(* CoDeSys 2.3.9.31 project: 3floor7(20131104).prx *)
(* Libraries: TcEIB.lbx 31.10.12 09:33:08, TcBaseBX.lbx 10.5.06 08:50:20, TcSystemBX.lbx 11.6.12 13:56:16, standard.lbx 5.12.03 08:02:30 *)

(* Task configuration *)
TASK Standard (PRIORITY := 0, INTERVAL := T#20ms);
	MAIN
END_TASK

(* Global variable list: main *)
VAR_GLOBAL


	bDarkOutside: BOOL;
	fb_KL6301_0: KL6301; (* EIB functonblock *)


	VITALNYA_HVAC: ROOM_HVAC;
	SPALNYA_HVAC: ROOM_HVAC;
	DYTJACHA_HVAC: ROOM_HVAC;
	KINO_HVAC:ROOM_HVAC;
	STUDIO_HVAC: ROOM_HVAC;
	KABINET_HVAC:ROOM_HVAC;

(*adresses for Temperatures from HDL panels *)
	vitalnya_T_EIB_addr: EIB_GROUP_ADDR:= (MAIN:=1, SUB_MAIN:=1, NUMBER:=0);
	kino_T_EIB_addr: EIB_GROUP_ADDR:= (MAIN:=1, SUB_MAIN:=2, NUMBER:=0);
	studio_T_EIB_addr: EIB_GROUP_ADDR:= (MAIN:=1, SUB_MAIN:=3, NUMBER:=0);
	kabinet_T_EIB_addr: EIB_GROUP_ADDR:= (MAIN:=1, SUB_MAIN:=4, NUMBER:=0);
	dytjacha_T_EIB_addr: EIB_GROUP_ADDR:= (MAIN:=1, SUB_MAIN:=5, NUMBER:=0);
	spalnya_T_EIB_addr: EIB_GROUP_ADDR:= (MAIN:=1, SUB_MAIN:=6, NUMBER:=0);
(*adresses for current speed and setpoint of cooling mode from HDL panels *)
	dytjacha_cooling_EIB_addr: EIB_GROUP_ADDR:= (MAIN:=1, SUB_MAIN:=1, NUMBER:=1);
	spalnya_cooling_EIB_addr: EIB_GROUP_ADDR:= (MAIN:=1, SUB_MAIN:=2, NUMBER:=1);
	vitalnya_cooling_EIB_addr: EIB_GROUP_ADDR:= (MAIN:=1, SUB_MAIN:=3, NUMBER:=1);
	kino_cooling_EIB_addr: EIB_GROUP_ADDR:= (MAIN:=1, SUB_MAIN:=4, NUMBER:=1);
	studio_cooling_EIB_addr: EIB_GROUP_ADDR:= (MAIN:=1, SUB_MAIN:=5, NUMBER:=1);
	kabinet_cooling_EIB_addr: EIB_GROUP_ADDR:= (MAIN:=1, SUB_MAIN:=6, NUMBER:=1);
(*adresses for current speed and setpoint of heating mode from HDL panels *)
	dytjacha_heating_EIB_addr: EIB_GROUP_ADDR:= (MAIN:=1, SUB_MAIN:=1, NUMBER:=2);
	spalnya_heating_EIB_addr: EIB_GROUP_ADDR:= (MAIN:=1, SUB_MAIN:=2, NUMBER:=2);
	vitalnya_heating_EIB_addr: EIB_GROUP_ADDR:= (MAIN:=1, SUB_MAIN:=3, NUMBER:=2);
	kino_heating_EIB_addr: EIB_GROUP_ADDR:= (MAIN:=1, SUB_MAIN:=4, NUMBER:=2);
	studio_heating_EIB_addr: EIB_GROUP_ADDR:= (MAIN:=1, SUB_MAIN:=5, NUMBER:=2);
	kabinet_heating_EIB_addr: EIB_GROUP_ADDR:= (MAIN:=1, SUB_MAIN:=6, NUMBER:=2);
(*adresses for current speed of fan mode from HDL panels *)
	dytjacha_fan_EIB_addr: EIB_GROUP_ADDR:= (MAIN:=1, SUB_MAIN:=1, NUMBER:=3);
	spalnya_fan_EIB_addr: EIB_GROUP_ADDR:= (MAIN:=1, SUB_MAIN:=2, NUMBER:=3);
	vitalnya_fan_EIB_addr: EIB_GROUP_ADDR:= (MAIN:=1, SUB_MAIN:=3, NUMBER:=3);
	kino_fan_EIB_addr: EIB_GROUP_ADDR:= (MAIN:=1, SUB_MAIN:=4, NUMBER:=3);
	studio_fan_EIB_addr: EIB_GROUP_ADDR:= (MAIN:=1, SUB_MAIN:=5, NUMBER:=3);
	kabinet_fan_EIB_addr: EIB_GROUP_ADDR:= (MAIN:=1, SUB_MAIN:=6, NUMBER:=3);


	shtory_kino_EIB_addr: EIB_GROUP_ADDR := (MAIN:=1, SUB_MAIN:=2, NUMBER:=30);
	tul_kino_EIB_addr: EIB_GROUP_ADDR := (MAIN:=1, SUB_MAIN:=2, NUMBER:=31);
	shtory_kabinet_EIB_addr: EIB_GROUP_ADDR := (MAIN:=1, SUB_MAIN:=4, NUMBER:=30);
	tul_kabinet_EIB_addr: EIB_GROUP_ADDR := (MAIN:=1, SUB_MAIN:=4, NUMBER:=31);
	shtory_spalnya_EIB_addr: EIB_GROUP_ADDR := (MAIN:=1, SUB_MAIN:=6, NUMBER:=31);
	tul_spalnya_EIB_addr: EIB_GROUP_ADDR := (MAIN:=1, SUB_MAIN:=6, NUMBER:=30);
	lift_spalnya_EIB_addr: EIB_GROUP_ADDR := (MAIN:=1, SUB_MAIN:=6, NUMBER:=29);
	tLongPress: TIME; (* затримка довгого натискання *)
	tOffDelay: TIME; (* затримка для відкладеного вимкнення *)
	ads_adr1: STRING;
	ads_adr2: STRING;
	ads_adr3: STRING;
	close_ads: ADSCLOSE;
	read_ads: ADSREAD;

	data1floor: ARRAY[0..20] OF SINT;
	data2floor: ARRAY[0..20] OF SINT;

	data1floor_prev: ARRAY[0..20] OF BYTE; (*попередні значення*)
	data2floor_prev: ARRAY[0..20] OF BYTE;

	moove_garderob				AT%MX0.0:BOOL;
	moove_tambur					AT%MX0.1:BOOL;
	moove_dytjacha					AT%MX0.2:BOOL;
	moove_spalnya					AT%MX0.3:BOOL;
	moove_korydor					AT%MX0.4:BOOL;
	moove_skhody					AT%MX0.5:BOOL;


END_VAR

(* Global variable list: physical *)
VAR_GLOBAL
	din1_1	AT %IX0.0:	BOOL;
	din1_2	AT %IX0.1:	BOOL;
	din1_3	AT %IX0.2:	BOOL;
	din1_4	AT %IX0.3:	BOOL;
	din1_5	AT %IX0.4:	BOOL;
	din1_6	AT %IX0.5:	BOOL;
	din1_7	AT %IX0.6:	BOOL;
	din1_8	AT %IX0.7:	BOOL;
	din2_1	AT %IX1.0:	BOOL;
	din2_2	AT %IX1.1:	BOOL;
	din2_3	AT %IX1.2:	BOOL;
	din2_4	AT %IX1.3:	BOOL;
	din2_5	AT %IX1.4:	BOOL;
	din2_6	AT %IX1.5:	BOOL;
	din2_7	AT %IX1.6:	BOOL;
	din2_8	AT %IX1.7:	BOOL;
	sw_garderob1	AT %IX2.0:	BOOL;
	sw_dytjacha1 	AT %IX2.1:	BOOL;
	sw_garderob2	AT %IX2.2:	BOOL;
	sw_dytjacha2		AT %IX2.3:	BOOL;
	sw_tambur3_2	AT %IX2.4:	BOOL;
	sw_korydor		AT %IX2.5:	BOOL;
	sw_tambur1		AT %IX2.6:	BOOL;
	din3_8			AT %IX2.7:	BOOL;
	sw_su2			AT %IX3.0:	BOOL;
	sw_spalnya3		AT %IX3.1:	BOOL;
	sw_su1			AT %IX3.2:	BOOL;
	sw_spalnya1		AT %IX3.3:	BOOL;
	sw_spalnya_balk	AT %IX3.4:	BOOL;
	sw_spalnya2		AT %IX3.5:	BOOL;
	sw_tambur3		AT %IX3.6:	BOOL;
	sw_spalnya4		AT %IX3.7:	BOOL;
(*dout1_1*)z_vitalnya	AT %QX0.0:	BOOL;
(*dout1_2*)z_spalnya	AT %QX0.1:	BOOL;
(*dout1_3*)z_kabinet	AT %QX0.2:	BOOL;
	dout1_4	AT %QX0.3:	BOOL;
(*dout1_5*)z_kino	AT %QX0.4:	BOOL;
	dout1_6	AT %QX0.5:	BOOL;
(*dout1_7*)z_dytjacha	AT %QX0.6:	BOOL;
	dout1_8	AT %QX0.7:	BOOL;
	dout2_1	AT %QX1.0:	BOOL;
	dout2_2	AT %QX1.1:	BOOL;
	dout2_3	AT %QX1.2:	BOOL;
	dout2_4	AT %QX1.3:	BOOL;
	dout2_5	AT %QX1.4:	BOOL;
	dout2_6	AT %QX1.5:	BOOL;
	dout2_7	AT %QX1.6:	BOOL;
	su3_vent	AT %QX1.7:	BOOL;
	dout3_1	AT %QX2.0:	BOOL;
	spalnya_kontrazhur	AT %QX2.1:	BOOL; (*c*)
	balkon				AT %QX2.2:	BOOL; (*c2*)
	dout3_4				AT %QX2.3:	BOOL;
	spalnya_kulbaba		AT %QX2.4:	BOOL;(*c3, c3a*)
	spalnya_kontrazhur_b	AT %QX2.5:	BOOL; (*c7*)
	spalnya_kontrazhur_l	AT %QX2.6:	BOOL; (*c4*)
	su3_stina			AT %QX2.7:	BOOL; (*c8*)
	(*dout4_1*)su3_pidsvitka 		AT %QX3.0:	BOOL;(*c10*)
	su3_bra				AT %QX3.1:	BOOL;(*c15*)
	su3_kontrazhur		AT %QX3.2:	BOOL;(*c9*)
	dytjacha				AT %QX3.3:	BOOL;(*c14*)
	su3_kontrazhur_k		AT %QX3.4:	BOOL; (*c11*)
	dytjacha_bra			AT %QX3.5:	BOOL; (*c15*)
	su3_lampa			AT %QX3.6:	BOOL; (*c12*)
	garderob			AT %QX3.7:	BOOL;
	(*dout5_1*)	garderob_serv		AT %QX4.0:	BOOL;
	bar					AT %QX4.1:	BOOL;(*c21*)
	korydor_skeli 		AT %QX4.2:	BOOL;(*c18*)
	choven				AT %QX4.3:	BOOL;(*c22*)
	korydor_svitlo		AT %QX4.4:	BOOL;(*c19*)
	fancoil_spalnya_low 	AT %QX4.5:	BOOL;
	korydor_lampa		AT %QX4.6:	BOOL;(*c20*)
	fancoil_spalnya_med	AT %QX4.7:	BOOL;
	(*dout6_1*)fancoil_spalnya_high	AT%QX5.0:BOOL;
	rozetky1				AT%QX5.1 :BOOL;
	fancoil_dytjacha_low	AT%QX5.2 :BOOL;
	rozetky2			 	AT%QX5.3 :BOOL;
	fancoil_dytjacha_med	AT%QX5.4:BOOL;
	rozetky3 				AT%QX5.5:BOOL;
	fancoil_dytjacha_high	AT%QX5.6:BOOL;
	rozetky4 				AT%QX5.7:BOOL;
	(*dout7_1*)rozetky5	AT%QX6.0:BOOL;
	tul_close 			AT%QX6.1 :BOOL;
	rozetky6	 			AT%QX6.2 :BOOL;
	tul_open	 			AT%QX6.3 :BOOL;
	shtory_close 			AT%QX6.4:BOOL;
	lift_down				AT%QX6.5:BOOL;
	shtory_open			AT%QX6.6:BOOL;
	lift_up	 			AT%QX6.7:BOOL;
(*dout8_1*) dytjacha_col AT%QX7.0:BOOL; (*тепла підлога*)
	serverna_col 		AT%QX7.1 :BOOL;
	freshbar_col 			AT%QX7.2 :BOOL;
	spalnya_col 		AT%QX7.3 :BOOL;
	korydor_col		 	AT%QX7.4:BOOL;
	su_col_pidloga 		AT%QX7.5:BOOL;
	su_col_stina		AT%QX7.6:BOOL;
	out88 AT%QX7.7:BOOL;
	out91 AT%QX8.0:BOOL;
	out92 AT%QX8.1 :BOOL;
	out93 AT%QX8.2 :BOOL;
	out94 AT%QX8.3 :BOOL;
	out95 AT%QX8.4:BOOL;
	out96 AT%QX8.5:BOOL;
	out97 AT%QX8.6:BOOL;
	out98 AT%QX8.7:BOOL;

	klapan_dytjacha		AT %QB10:	INT;
	klapan_spalnya		AT %QB12:	INT;
	KL4414_3_Out		AT %QB14:	INT;
	klapan_vitalnya		AT %QB16:	INT;
(*light sensors*)
	iLight_N			AT %IB20:INT;
	iLight_W			AT %IB22:INT;
	iLight_S			AT %IB28:INT;
	iLight_E			AT %IB26:INT;

	KL6301_IN_0 AT %IB4: ARRAY[1..24] OF BYTE;
	KL6301_OUT_0 AT %QB34: ARRAY[1..24] OF BYTE;

	temp_tambur	AT %IB30: INT;(*тепла підлога*)
	temp_su		AT %IB32: INT;(*тепла підлога*)
	temp_spalnya	AT %IB34: INT;(*тепла підлога*)
	iT_out			AT %IB36:INT; (*зовнішня температура*)

END_VAR

(* Data type *)
TYPE ROOM_HVAC :
STRUCT

	heat_mode: STRING;
	heat_speed: USINT;

	cur_t:REAL;
	t_ust:REAL;

	fancoil_speed:SINT;
	klapan:WORD;

	tepla_pidloga:BOOL;

	zaslinka:BOOL;


END_STRUCT
END_TYPE

(* POU MAIN, ST *)
PROGRAM MAIN
VAR
	fbTimer: TON;
	fbRTC: RTC;
	i:INT;
	system_time:timestruct;
	fbDarkTimeCorrection : TP;


END_VAR
(*Parameters*)
	tLongPress:=t#500ms; (*затримка довгого натискання*)
	tOffDelay:=t#5m; (*затримка для відкладеного вимкнення*)

	ads_adr1:='10.0.5.61.1.1';
	ads_adr2:='10.0.5.62.1.1';
	ads_adr3:='10.0.5.63.1.1';

fbTimer(PT:=t#1s,IN:=NOT fbTimer.Q);

IF fbTimer.Q OR SYSTEMTASKINFOARR[1].firstCycle  THEN
	fbRTC;
END_IF

system_time:=DT_TO_SYSTEMTIME(fbRTC.CDT);
data1floor[4]:=WORD_TO_BYTE(system_time.wHour);
data1floor[5]:=WORD_TO_BYTE(system_time.wMinute);
data2floor[9]:=WORD_TO_BYTE(system_time.wHour);
data2floor[10]:=WORD_TO_BYTE(system_time.wMinute);

fbDarkTimeCorrection(IN:=iLight_N<1000 AND  iLight_W <1000 AND iLight_S <1000 AND iLight_E <1000, PT:=t#40m);
IF iLight_N<1000 AND  iLight_W <1000 AND iLight_S <1000 AND iLight_E <1000  AND NOT fbDarkTimeCorrection.q THEN
	bDarkOutside:=TRUE;
ELSE
	bDarkOutside:=FALSE;
END_IF

data2floor[6].1:=bDarkOutside;
data1floor[2].6:=bDarkOutside;
(*EIB init*)
EIB;
(*Світло*)
light;
shtory;
(*тепло*)
heat;
ADS_write;
END_PROGRAM

(* POU EIB, ST *)
PROGRAM EIB
VAR
	i:INT:=0;
	POWER: EIB_BIT_REC;
	fb_temp_read: EIB_2OCTET_FLOAT_REC;
	fb_setpoint_read:EIB_8BIT_UNSIGN_REC;



	temp:INT;
	inc: BYTE;		(*increment for temperature read cycles*)
END_VAR
(*EIB*)
fb_KL6301_0.iMode:=1;
CASE i OF
0:	(* EIB Address 2.3.4 *)
	fb_KL6301_0.EIB_PHYS_ADDR.Area:=15;
	fb_KL6301_0.EIB_PHYS_ADDR.Line:=15;
	fb_KL6301_0.EIB_PHYS_ADDR.Device:=15;
	(* Filter 1 *)
	fb_KL6301_0.EIB_GROUP_FILTER[1].GROUP_ADDR.MAIN:=1;
	fb_KL6301_0.EIB_GROUP_FILTER[1].GROUP_ADDR.SUB_MAIN:=1;
	fb_KL6301_0.EIB_GROUP_FILTER[1].GROUP_ADDR.NUMBER:=0;
	fb_KL6301_0.EIB_GROUP_FILTER[1].GROUP_LEN:=31;
	(* Filter 2*)
	fb_KL6301_0.EIB_GROUP_FILTER[2].GROUP_ADDR.MAIN:=1;
	fb_KL6301_0.EIB_GROUP_FILTER[2].GROUP_ADDR.SUB_MAIN:=2;
	fb_KL6301_0.EIB_GROUP_FILTER[2].GROUP_ADDR.NUMBER:=0;
	fb_KL6301_0.EIB_GROUP_FILTER[2].GROUP_LEN:=31;
	(* Filter 3*)
	fb_KL6301_0.EIB_GROUP_FILTER[3].GROUP_ADDR.MAIN:=1;
	fb_KL6301_0.EIB_GROUP_FILTER[3].GROUP_ADDR.SUB_MAIN:=3;
	fb_KL6301_0.EIB_GROUP_FILTER[3].GROUP_ADDR.NUMBER:=0;
	fb_KL6301_0.EIB_GROUP_FILTER[3].GROUP_LEN:=31;
	(* Filter 4 *)
	fb_KL6301_0.EIB_GROUP_FILTER[4].GROUP_ADDR.MAIN:=1;
	fb_KL6301_0.EIB_GROUP_FILTER[4].GROUP_ADDR.SUB_MAIN:=4;
	fb_KL6301_0.EIB_GROUP_FILTER[4].GROUP_ADDR.NUMBER:=0;
	fb_KL6301_0.EIB_GROUP_FILTER[4].GROUP_LEN:=31;
	(* Filter 5*)
	fb_KL6301_0.EIB_GROUP_FILTER[5].GROUP_ADDR.MAIN:=1;
	fb_KL6301_0.EIB_GROUP_FILTER[5].GROUP_ADDR.SUB_MAIN:=5;
	fb_KL6301_0.EIB_GROUP_FILTER[5].GROUP_ADDR.NUMBER:=0;
	fb_KL6301_0.EIB_GROUP_FILTER[5].GROUP_LEN:=31;
	(* Filter 6*)
	fb_KL6301_0.EIB_GROUP_FILTER[6].GROUP_ADDR.MAIN:=1;
	fb_KL6301_0.EIB_GROUP_FILTER[6].GROUP_ADDR.SUB_MAIN:=6;
	fb_KL6301_0.EIB_GROUP_FILTER[6].GROUP_ADDR.NUMBER:=0;
	fb_KL6301_0.EIB_GROUP_FILTER[6].GROUP_LEN:=31;
	(* Filter 7*)
	fb_KL6301_0.EIB_GROUP_FILTER[7].GROUP_ADDR.MAIN:=1;
	fb_KL6301_0.EIB_GROUP_FILTER[7].GROUP_ADDR.SUB_MAIN:=7;
	fb_KL6301_0.EIB_GROUP_FILTER[7].GROUP_ADDR.NUMBER:=0;
	fb_KL6301_0.EIB_GROUP_FILTER[7].GROUP_LEN:=31;
(*	(* Filter 8*)
	fb_KL6301_0.EIB_GROUP_FILTER[8].GROUP_ADDR.MAIN:=1;
	fb_KL6301_0.EIB_GROUP_FILTER[8].GROUP_ADDR.SUB_MAIN:=8;
	fb_KL6301_0.EIB_GROUP_FILTER[8].GROUP_ADDR.NUMBER:=0;
	fb_KL6301_0.EIB_GROUP_FILTER[8].GROUP_LEN:=31;*)

	fb_KL6301_0.bActivate :=TRUE; 	(*Start EIB Functionblock*)
	IF fb_KL6301_0.bReady THEN	(*Wait until the fb is ready *)
		IF NOT fb_KL6301_0.bError THEN
			i:=1;  (* EIB functionblock is now ready to send and receive *)
		ELSE
			i:=100; (* EIB ERROR*)
		END_IF
	END_IF
1:	;
100:	;(*ERROR EIB*)
END_CASE

fb_KL6301_0(
	idx:=1,								(* for every KL6301 an other idx number
										Example KL6301 terminal 1 - idx=1 , KL6301 termnal 2 -idx=3,... max. 64 *)
	KL6301_IN:=KL6301_IN_0,				(* Terminal variable - address IN *)
	KL6301_OUT:=KL6301_OUT_0 );			(* Terminal variable - address OUT *)


fb_temp_read(Group_Address:=vitalnya_T_EIB_addr, strData_Rec:=fb_KL6301_0.str_Data_Rec);
fb_temp_read(Group_Address:=kino_T_EIB_addr, strData_Rec:=fb_KL6301_0.str_Data_Rec);
fb_temp_read(Group_Address:=studio_T_EIB_addr, strData_Rec:=fb_KL6301_0.str_Data_Rec);
fb_temp_read(Group_Address:=kabinet_T_EIB_addr, strData_Rec:=fb_KL6301_0.str_Data_Rec);
fb_temp_read(Group_Address:=dytjacha_T_EIB_addr, strData_Rec:=fb_KL6301_0.str_Data_Rec);
fb_temp_read(Group_Address:=spalnya_T_EIB_addr, strData_Rec:=fb_KL6301_0.str_Data_Rec);

IF  fb_KL6301_0.GroupReceive.NUMBER=0 THEN
	IF fb_KL6301_0.GroupReceive.SUB_MAIN=vitalnya_T_EIB_addr.SUB_MAIN THEN  VITALNYA_HVAC.cur_t:=(fb_temp_read.rData); END_IF
	IF fb_KL6301_0.GroupReceive.SUB_MAIN=kino_T_EIB_addr.SUB_MAIN THEN  KINO_HVAC.cur_t:=(fb_temp_read.rData);END_IF
	IF fb_KL6301_0.GroupReceive.SUB_MAIN=studio_T_EIB_addr.SUB_MAIN THEN  STUDIO_HVAC.cur_t:=(fb_temp_read.rData);END_IF
	IF fb_KL6301_0.GroupReceive.SUB_MAIN=kabinet_T_EIB_addr.SUB_MAIN THEN  KABINET_HVAC.cur_t:=(fb_temp_read.rData);END_IF
	IF fb_KL6301_0.GroupReceive.SUB_MAIN=dytjacha_T_EIB_addr.SUB_MAIN THEN  DYTJACHA_HVAC.cur_t:=(fb_temp_read.rData);END_IF
	IF fb_KL6301_0.GroupReceive.SUB_MAIN=spalnya_T_EIB_addr.SUB_MAIN THEN  SPALNYA_HVAC.cur_t:=(fb_temp_read.rData);END_IF
END_IF


fb_setpoint_read(Group_Address:=vitalnya_cooling_EIB_addr, strData_Rec:=fb_KL6301_0.str_Data_Rec);
fb_setpoint_read(Group_Address:=kino_cooling_EIB_addr, strData_Rec:=fb_KL6301_0.str_Data_Rec);
fb_setpoint_read(Group_Address:=studio_cooling_EIB_addr, strData_Rec:=fb_KL6301_0.str_Data_Rec);
fb_setpoint_read(Group_Address:=kabinet_cooling_EIB_addr, strData_Rec:=fb_KL6301_0.str_Data_Rec);
fb_setpoint_read(Group_Address:=dytjacha_cooling_EIB_addr, strData_Rec:=fb_KL6301_0.str_Data_Rec);
fb_setpoint_read(Group_Address:=spalnya_cooling_EIB_addr, strData_Rec:=fb_KL6301_0.str_Data_Rec);

fb_setpoint_read(Group_Address:=vitalnya_heating_EIB_addr, strData_Rec:=fb_KL6301_0.str_Data_Rec);
fb_setpoint_read(Group_Address:=kino_heating_EIB_addr, strData_Rec:=fb_KL6301_0.str_Data_Rec);
fb_setpoint_read(Group_Address:=studio_heating_EIB_addr, strData_Rec:=fb_KL6301_0.str_Data_Rec);
fb_setpoint_read(Group_Address:=kabinet_heating_EIB_addr, strData_Rec:=fb_KL6301_0.str_Data_Rec);
fb_setpoint_read(Group_Address:=dytjacha_heating_EIB_addr, strData_Rec:=fb_KL6301_0.str_Data_Rec);
fb_setpoint_read(Group_Address:=spalnya_heating_EIB_addr, strData_Rec:=fb_KL6301_0.str_Data_Rec);

fb_setpoint_read(Group_Address:=vitalnya_fan_EIB_addr, strData_Rec:=fb_KL6301_0.str_Data_Rec);
fb_setpoint_read(Group_Address:=kino_fan_EIB_addr, strData_Rec:=fb_KL6301_0.str_Data_Rec);
fb_setpoint_read(Group_Address:=studio_fan_EIB_addr, strData_Rec:=fb_KL6301_0.str_Data_Rec);
fb_setpoint_read(Group_Address:=kabinet_fan_EIB_addr, strData_Rec:=fb_KL6301_0.str_Data_Rec);
fb_setpoint_read(Group_Address:=dytjacha_fan_EIB_addr, strData_Rec:=fb_KL6301_0.str_Data_Rec);
fb_setpoint_read(Group_Address:=spalnya_fan_EIB_addr, strData_Rec:=fb_KL6301_0.str_Data_Rec);



(*CASE fb_KL6301_0.GroupReceive.SUB_MAIN OF
(*Вітальня 1го поверху*)
1:	CASE fb_KL6301_0.GroupReceive.NUMBER OF
		100:	POWER(Group_Address:=vitalnya_EIB_addr, strData_Rec:=fb_KL6301_0.str_Data_Rec ); (*З самого початку було вимкнення якщо на адресу приходив нуль*)

			IF POWER.bData=1 THEN
				VITALNYA_HVAC.heat_mode:='ON';

			END_IF;
			IF POWER.bData =0 THEN
				VITALNYA_HVAC.heat_mode:='OFF';
			END_IF;

		1: VITALNYA_HVAC.heat_mode:='COOL';
		2: VITALNYA_HVAC.heat_mode:='HEAT';
		3: VITALNYA_HVAC.heat_mode:='FAN'; (* вмикається режим FAN.  повне закриття клапана *)
		4: VITALNYA_HVAC.heat_speed:=3; (*high*)
		5: VITALNYA_HVAC.heat_speed:=2; (*med*)
		6: VITALNYA_HVAC.heat_speed:=1; (*low*)
	END_CASE;
(*Кінотеатр*)
2: 	CASE fb_KL6301_0.GroupReceive.NUMBER OF
		100:	POWER(Group_Address:=kino_EIB_addr, strData_Rec:=fb_KL6301_0.str_Data_Rec );

			IF POWER.bData=1 THEN
				KINO_HVAC.heat_mode:='ON';

			END_IF;
			IF POWER.bData =0 THEN
				KINO_HVAC.heat_mode:='OFF';
			END_IF;

		1: KINO_HVAC.heat_mode:='COOL';
		2: KINO_HVAC.heat_mode:='HEAT';
		3: KINO_HVAC.heat_mode:='FAN'; (* вмикається режим FAN.  повне закриття клапана *)
		4: KINO_HVAC.heat_speed:=3; (*high*)
		5: KINO_HVAC.heat_speed:=2; (*med*)
		6: KINO_HVAC.heat_speed:=1; (*low*)
	END_CASE;
(*Студія*)
3: 	CASE fb_KL6301_0.GroupReceive.NUMBER OF
		100:	POWER(Group_Address:=studio_EIB_addr, strData_Rec:=fb_KL6301_0.str_Data_Rec );

			IF POWER.bData=1 THEN
				STUDIO_HVAC.heat_mode:='ON';

			END_IF;
			IF POWER.bData =0 THEN
				STUDIO_HVAC.heat_mode:='OFF';
			END_IF;

		1: STUDIO_HVAC.heat_mode:='COOL';
		2: STUDIO_HVAC.heat_mode:='HEAT';
		3: STUDIO_HVAC.heat_mode:='FAN'; (* вмикається режим FAN.  повне закриття клапана *)
		4: STUDIO_HVAC.heat_speed:=3; (*high*)
		5: STUDIO_HVAC.heat_speed:=2; (*med*)
		6: STUDIO_HVAC.heat_speed:=1; (*low*)
	END_CASE;
(*Кабінет*)
4:	CASE fb_KL6301_0.GroupReceive.NUMBER OF
		100:	POWER(Group_Address:=kabinet_EIB_addr, strData_Rec:=fb_KL6301_0.str_Data_Rec );

			IF POWER.bData=1 THEN
				KABINET_HVAC.heat_mode:='ON';

			END_IF;
			IF POWER.bData =0 THEN
				KABINET_HVAC.heat_mode:='OFF';
			END_IF;

		1: KABINET_HVAC.heat_mode:='COOL';
		2: KABINET_HVAC.heat_mode:='HEAT';
		3: KABINET_HVAC.heat_mode:='FAN'; (* вмикається режим FAN.  повне закриття клапана *)
		4: KABINET_HVAC.heat_speed:=3; (*high*)
		5: KABINET_HVAC.heat_speed:=2; (*med*)
		6: KABINET_HVAC.heat_speed:=1; (*low*)
	END_CASE;
(*Дитяча*)
5: 	CASE fb_KL6301_0.GroupReceive.NUMBER OF
		100:	POWER(Group_Address:=dytjacha_EIB_addr, strData_Rec:=fb_KL6301_0.str_Data_Rec );

			IF POWER.bData=1 THEN
				DYTJACHA_HVAC.heat_mode:='ON';

			END_IF;
			IF POWER.bData =0 THEN
				DYTJACHA_HVAC.heat_mode:='OFF';
			END_IF;

		1: DYTJACHA_HVAC.heat_mode:='COOL';
		2: DYTJACHA_HVAC.heat_mode:='HEAT';
		3: DYTJACHA_HVAC.heat_mode:='FAN'; (* вмикається режим FAN.  повне закриття клапана *)
		4: DYTJACHA_HVAC.heat_speed:=3; (*high*)
		5: DYTJACHA_HVAC.heat_speed:=2; (*med*)
		6: DYTJACHA_HVAC.heat_speed:=1; (*low*)
	END_CASE
(*Спальня*)
6: CASE fb_KL6301_0.GroupReceive.NUMBER OF
		100:	POWER(Group_Address:=spalnya_EIB_addr, strData_Rec:=fb_KL6301_0.str_Data_Rec );

			IF POWER.bData=1 THEN
				SPALNYA_HVAC.heat_mode:='ON';

			END_IF;
			IF POWER.bData =0 THEN
				SPALNYA_HVAC.heat_mode:='OFF';
			END_IF;

		1: SPALNYA_HVAC.heat_mode:='COOL';
		2: SPALNYA_HVAC.heat_mode:='HEAT';
		3: SPALNYA_HVAC.heat_mode:='FAN'; (* вмикається режим FAN.  повне закриття клапана *)
		4: SPALNYA_HVAC.heat_speed:=3; (*high*)
		5: SPALNYA_HVAC.heat_speed:=2; (*med*)
		6: SPALNYA_HVAC.heat_speed:=1; (*low*)
	END_CASE;
END_CASE;

*)
END_PROGRAM

(* POU LIGHT, ST *)
PROGRAM LIGHT
VAR
	tambur1, tambur2,tambur3 : SWITCH;
	korydor : SWITCH;
	spalnya1,spalnya2, spalnya_balk:SWITCH;
	dytjacha1,dytjacha2  : SWITCH;
	su1 : SWITCH;
	su2: SWITCH;
	garderob1, garderob2 : SWITCH;

	tLightWindow: TIME;		(*Час, який світло світиться після спрацювання сенсора руху*)

	VENT_TIMER: TOF;		(*Таймер роботи вентилятора в пустому туалеті*)
	vent_timer_start: R_TRIG;
	test: BOOL;

	CHOVEN_TIMER: TOF;	(*Таймер роботи світильника на човні*)

	bChovenTimerOverride: SEMA;		(*Перевага вимикача над таймером*)
	bGarderobTimerOverride: SEMA;		(*Перевага вимикача над таймером*)
	KORYDOR_TIMER: TOF;		(*Таймер роботи світла в коридорі*)
	KORYDOR_F: F_TRIG;
	GARDEROB_TIMER: TOF;		(*Таймер роботи світла в гардеробі*)
	GARDEROB_F: F_TRIG;		(*Спрацювання сенсора руху в гардеробі*)
	KORYDOR_SEMA:SEMA;
	su_light: BOOL;
	vymykach3: BOOL;
END_VAR
tLightWindow:=t#60s;
(*Опитування вимикачів*)
tambur1(IN:=sw_tambur1);
tambur2(IN:=sw_tambur3_2);
tambur3(IN:=sw_tambur3);



spalnya1(IN:=sw_spalnya1 XOR sw_spalnya4);
spalnya2(IN:=sw_spalnya2 XOR sw_spalnya3);
spalnya_balk(IN:=sw_spalnya_balk);

dytjacha1(IN:=sw_dytjacha1);
dytjacha2(IN:=sw_dytjacha2);

su1(IN:=sw_su1);
su2(IN:=sw_su2);




(*запуск вечірніх таймерів світла*)
IF bDarkOutside THEN
	CHOVEN_TIMER(IN:= NOT moove_skhody, PT:= tLightWindow);
	KORYDOR_TIMER(IN:= NOT moove_korydor, PT:= tLightWindow);

END_IF

(*обробка сигналів вимикачів та таймерів*)
IF tambur1.short THEN bar:= NOT bar; END_IF


(*Відправка на 1,2 поверхи значення вимикача*)
data2floor[6].0:=sw_tambur3_2;
data1floor[2].1:=sw_tambur3_2;

IF tambur3.short THEN
	choven:= NOT choven;
END_IF
bChovenTimerOverride(CLAIM:=  NOT moove_skhody, RELEASE:=tambur3.short);
IF  bChovenTimerOverride.BUSY AND CHOVEN_TIMER.ET<>t#0ms THEN
	choven:=CHOVEN_TIMER.Q;
END_IF


korydor(IN:=sw_korydor);

korydor_lampa:=KORYDOR_TIMER.Q;
korydor_skeli:=korydor_lampa;
KORYDOR_F(clk:=korydor_timer.Q);
KORYDOR_SEMA(CLAIM:=(NOT korydor_svitlo AND korydor.short ), RELEASE:=(korydor_svitlo AND korydor.short) OR KORYDOR_f.Q);
korydor_svitlo:=KORYDOR_SEMA.BUSY;
IF spalnya1.short THEN spalnya_kulbaba:=NOT spalnya_kulbaba; END_IF
IF spalnya2.short THEN spalnya_kontrazhur:= NOT spalnya_kontrazhur; END_IF
spalnya_kontrazhur_b:=spalnya_kontrazhur;
spalnya_kontrazhur_l:=spalnya_kontrazhur;

IF spalnya_balk.short THEN balkon:=NOT balkon; END_IF

IF dytjacha1.short THEN dytjacha:= NOT dytjacha; END_IF
IF dytjacha2.short THEN dytjacha_bra:= NOT dytjacha_bra; END_IF

IF su2.short THEN	su3_bra:= NOT su3_bra; END_IF
	su3_lampa:= su3_bra;
	su3_kontrazhur:=su3_lampa;

IF su2.long THEN	su3_stina:= NOT su3_stina; END_IF
	su3_kontrazhur_k:= su3_stina;

IF su1.long THEN su3_vent:= NOT su3_vent; END_IF
IF su1.short THEN su3_pidsvitka:= NOT su3_pidsvitka; END_IF
(*IF su1.short AND NOT su3_vent THEN su3_vent:=TRUE; END_IF; *) (*вмикання вентилятора разом зі світлом*)

(*
вмикання вентилятора на деякий час після того, як вимикається все світло у ванній

su_light:=su3_stina OR su3_kontrazhur OR su3_bra OR su3_pidsvitka;

vent_timer_start(CLK:=NOT su_light );
VENT_TIMER(PT:=tOffDelay,IN:=vent_timer_start.Q);
IF NOT su_light THEN
	su3_vent:= VENT_TIMER.Q;
END_IF
*)


garderob1(IN:=sw_garderob1);
garderob2(IN:=sw_garderob2);
GARDEROB_F(CLK:=moove_garderob);
GARDEROB_TIMER(IN:= GARDEROB_F.Q, PT:= tLightWindow*2);

IF garderob2.short THEN garderob_serv := NOT garderob_serv; END_IF

bGarderobTimerOverride(CLAIM:=  (NOT moove_garderob OR (NOT garderob AND garderob1.short)), RELEASE:=  (garderob AND  garderob1.short) );
garderob:=bGarderobTimerOverride.BUSY;
END_PROGRAM

(* POU Vymykachi/SWITCH, ST *)
FUNCTION_BLOCK SWITCH
VAR_INPUT
	IN:BOOL;
	SHORT_OFF_DELAY, LONG_OFF_DELAY: TIME; (*час затримки вимкнення по короткому та довгому натисненню*)
END_VAR
VAR_OUTPUT
	short, long:BOOL;
END_VAR
VAR
	tChas: TIME; (*час доки кнопка натиснена*)
	TIMER: TON; (*таймер час натискання*)
	bPressed:BOOL;
	turn_off_long: BOOL;
	start_l, start_s:BOOL;
	bStan: BOOL:=FALSE;
END_VAR
short:=FALSE;
long:=FALSE;
TIMER(IN:=IN AND bStan, PT:=t#10s);
IF IN AND bStan THEN
	tChas:=timer.ET;
	bPressed:=TRUE;
ELSE
	bPressed:=FALSE;
END_IF;

IF NOT IN AND NOT bStan THEN
	tChas:=t#0ms;
END_IF;

IF bStan AND NOT IN THEN
	IF tChas <tLongPress THEN
		short:=TRUE;
	END_IF;
	IF tChas>=tLongPress THEN
		long:=TRUE;
	END_IF;
END_IF;
bStan := IN;
END_FUNCTION_BLOCK

(* POU shtory, ST *)
PROGRAM shtory
VAR
	inc1, inc: UINT;
	impulse: BOOL;
	last_move: UINT;
	impulse1: BOOL;
	last_move1: UINT;
	lift_move_dir, lift_move: BOOL;
	rising1: BOOL;
	falling1: BOOL;
	rising2: BOOL;
	falling2: BOOL;
	panel_shtory_move, panel_tul_move, panel_lift_move:BOOL;
	eib_shtory, eib_tul, eib_lift: EIB_BIT_REC;
	eib_shtory_kino, eib_tul_kino: EIB_BIT_REC; (*ловлять в мережі смартбаса телеграмки для штор і тюлей*)
	eib_shtory_kabinet, eib_tul_kabinet: EIB_BIT_REC;
	(*таймери для формування керуючих імпульсів*)
	timer_shtory_move, timer_shtory_stop,timer_tul_move, timer_tul_stop, move_lift_up, move_lift_down: TP;
	counter:CTU;
	shtory_move: BOOL;
	tul_move: BOOL;
	bBlock:BOOL;
	darkness_shtory_move: TP;
	btest: BOOL;
END_VAR
bBlock:=FALSE;
IF MAIN.fbRTC.stSystemTime.wHour=8 AND MAIN.fbRTC.stSystemTime.wMinute=0 AND MAIN.fbRTC.stSystemTime.wSecond<22 THEN
	bBlock:=TRUE;
	lift_down:=TRUE;
	lift_up:=FALSE;
	lift_move_dir:=FALSE;
	shtory_open:=TRUE;
	shtory_close:=FALSE;
	tul_open:=FALSE;
	tul_close:=TRUE;

ELSE
	(*детекція відсутності фронтів*)
	IF LIGHT.spalnya1.long = impulse THEN
		rising1:=0;
		falling1:=0;
	END_IF;

	IF LIGHT.spalnya2.long = impulse1  THEN
		rising2:=0;
		falling2:=0;
	END_IF;

	(*якщо клавіші довго  натиснені одночасно, то рухати ліфт, якщо довго і окремо - штори*)
	IF ( (LIGHT.spalnya1.long AND LIGHT.spalnya2.long) OR panel_lift_move)  AND NOT( move_lift_up.Q OR  move_lift_down.Q)  THEN
		lift_move:=1;
		lift_move_dir:= NOT lift_move_dir;
	ELSE

		(*ловим передній фронт довгого натискання першої клавіші*)
		IF LIGHT.spalnya1.long AND NOT impulse  AND NOT LIGHT.spalnya2.long THEN
			rising1:=1;
			falling1:=0;
		END_IF;

		(*задній фронт*)
		IF NOT LIGHT.spalnya1.long AND  impulse AND NOT LIGHT.spalnya2.long  THEN
			falling1:=1;
			rising1:=0;
		END_IF;

		(*ловим передній фронт довгого натискання другої клавіші*)
		IF LIGHT.spalnya2.long AND NOT impulse1 AND NOT LIGHT.spalnya1.long  THEN
			rising2:=1;
			falling2:=0;
		END_IF;

		(*ловим задній фронт довгого натискання другої клавіші*)
		IF NOT LIGHT.spalnya2.long AND  impulse1 AND NOT LIGHT.spalnya1.long THEN
			falling2:=1;
			rising2:=0;
		END_IF
	END_IF
	(*команди шторам та ліфту з панелей смартбаса*)
	eib_shtory(Group_Address:=shtory_spalnya_EIB_addr, strData_Rec:=fb_KL6301_0.str_Data_Rec);
	eib_tul(Group_Address:=tul_spalnya_EIB_addr, strData_Rec:=fb_KL6301_0.str_Data_Rec);
	eib_lift(Group_Address:=lift_spalnya_EIB_addr, strData_Rec:=fb_KL6301_0.str_Data_Rec);

	eib_shtory_kino(Group_Address:=shtory_kino_EIB_addr, strData_Rec:=fb_KL6301_0.str_Data_Rec);
	eib_tul_kino(Group_Address:=tul_kino_EIB_addr, strData_Rec:=fb_KL6301_0.str_Data_Rec);

	eib_shtory_kabinet(Group_Address:=shtory_kabinet_EIB_addr, strData_Rec:=fb_KL6301_0.str_Data_Rec);
	eib_tul_kabinet(Group_Address:=tul_kabinet_EIB_addr, strData_Rec:=fb_KL6301_0.str_Data_Rec);

	IF NOT eib_shtory_kabinet.bDataReceive THEN data2floor[7].0:=NOT data2floor[7].0; END_IF
	IF NOT eib_tul_kabinet.bDataReceive THEN data2floor[7].1:=NOT data2floor[7].1; END_IF
	IF NOT eib_shtory_kino.bDataReceive THEN data2floor[7].2:=NOT data2floor[7].2; END_IF
	IF NOT eib_tul_kino.bDataReceive THEN data2floor[7].3:=NOT data2floor[7].3; END_IF

	panel_tul_move:= NOT eib_tul.bDataReceive;
	panel_shtory_move:= NOT eib_shtory.bDataReceive;
	panel_lift_move:=NOT eib_lift.bDataReceive;


	shtory_move:= LIGHT.spalnya1.long OR panel_shtory_move;
	tul_move:= LIGHT.spalnya2.long OR panel_tul_move;



	(*формування імпульсів для керування шторами, тюлями та ліфтом*)
	timer_shtory_move(IN:=shtory_move, PT:=t#500ms);
	timer_shtory_stop(IN:=shtory_move , PT:=t#500ms);
	timer_tul_move(IN:=tul_move  , PT:=t#500ms);
	timer_tul_stop(IN:=tul_move , PT:=t#500ms);

	move_lift_up(IN:=lift_move AND lift_move_dir , PT:=t#20s,Q=>lift_up);
	move_lift_down(IN:=lift_move AND NOT lift_move_dir, PT:=t#20s, Q=>lift_down);



	darkness_shtory_move(IN:=bDarkOutside, PT:=t#15s);
	IF darkness_shtory_move.Q THEN
		shtory_open:=FALSE;
		shtory_close:=TRUE;
		tul_open:=FALSE;
		tul_close:=TRUE;
		bBlock:=TRUE;
	END_IF


	IF NOT bBlock THEN
		IF NOT (LIGHT.spalnya1.long AND LIGHT.spalnya2.long) THEN (*якщо не засік довгого затискання двох клавіш (ліфт не рухається) - рухати штори *)

		(*вибір рухати чи зупинити  штори*)
			IF shtory_move   THEN
				inc:=inc+1;
			END_IF;
			IF inc>2 THEN inc:=1; END_IF;

			(*вибір рухати чи зупинити  тюль*)
			IF tul_move THEN
				inc1:=inc1+1;
			END_IF;
			IF inc1>2 THEN inc1:=1; END_IF;

			CASE inc OF

				1:
				shtory_open:=timer_shtory_move.Q; (*відкривати*)
				shtory_close:= 0;
				last_move:=inc;

				2:
				shtory_close:=timer_shtory_move.Q;(*закривати*)
				shtory_open:= 0;
				last_move:=inc;

			END_CASE;

			CASE inc1 OF

				1:
				tul_open:=timer_tul_move.Q; (*відкривати*)
				tul_close:= 0;
				last_move1:=inc;
				2:
				tul_close:=timer_tul_move.Q;(*закривати*)
				tul_open:= 0;
				last_move1:=inc;

			END_CASE;

		END_IF;
	END_IF

	(*запам'ятовування стану довгого натискання для детекції фронтів*)

	impulse:=LIGHT.spalnya1.long;
	impulse1:=LIGHT.spalnya2.long;

	 lift_move:= 0;
END_IF
END_PROGRAM

(* POU HVAC/heat, ST *)
PROGRAM heat
VAR PERSISTENT

	t_out, t_out_avg_day, t_out_avg_10day:REAL;
	measures_this_day, meashured_days:INT;
	day_sum, ten_day_sum:REAL;
END_VAR


VAR
	temp_measure:TOF; (*таймер задає частоту замірів температури*)
	(*актуальна та попередня температури*)
	t_tambur, t_tamburPrev: REAL;
	t_su, t_suPrev: REAL;
	t_spalnya, t_spalnyaPrev: REAL;
	t_outPrev:REAL;
	(*мінімум та максимум температур теплих підлог*)
	t_max: REAL;
	t_min: REAL;
	(*різниця між поперднім та актуальним значенням температури*)
	delta_out, delta_tambur, delta_su, delta_spalnya: REAL;

	i: INT:=0;
	fbRetryCounter:CTU;
	iRetryCounter:INT;
	(*використовуються для знаходження середньої температури при ініціації*)
	t_tambur_sum: REAL;
	t_su_sum: REAL;
	t_spalnya_sum: REAL;
	t_out_sum: REAL;
	retry: BOOL:=TRUE;		(*переміряти температуру*)
END_VAR
(*фільтр показань сенсорів температури*)
CASE i OF
0..500: init;
ELSE
	IF retry THEN
		temp_measure.PT:=t#2s;

	ELSE temp_measure.PT:=t#5m;
	END_IF
	IF retry THEN
		IF iRetryCounter >5 THEN iRetryCounter:=0; i:=0; ELSE iRetryCounter:=iRetryCounter+1; END_IF;
	END_IF;
	temp_measure( IN:=NOT temp_measure.q); (*перевіряти температуру кожні 20 хв*)


IF NOT temp_measure.Q THEN

	delta_spalnya:=ABS(t_spalnyaPrev-temp_spalnya*0.1);
	delta_su:=ABS(t_suPrev-temp_su*0.1);
	delta_tambur:=ABS(t_tamburPrev-temp_tambur*0.1);
	delta_out:=ABS(t_outPrev-iT_out*0.1);
	retry:=FALSE;
	IF delta_spalnya<1 THEN
		t_spalnya:= temp_spalnya * 0.1;
	ELSE
		t_spalnya:=t_spalnyaPrev;
		retry:=TRUE;
	END_IF

	IF delta_su<1 THEN
		t_su:= temp_su * 0.1;
	ELSE
		t_su:=t_suPrev;
		retry:=TRUE;
	END_IF

	IF delta_tambur<1 THEN
		t_tambur:= temp_tambur * 0.1;
	ELSE
		t_tambur:=t_tamburPrev;
		retry:=TRUE;
	END_IF

	IF delta_out<01 THEN
		t_out:= iT_out* 0.1;
	ELSE
		t_out:=t_outPrev;
		retry:=TRUE;
	END_IF

	t_spalnyaPrev:=t_spalnya;
	t_suPrev:=t_su;
	t_tamburPrev:=t_tambur;
	t_outPrev:=t_out;

END_IF
END_CASE

(*CASE MAIN.fbRTC.stSystemTime.wSecond OF*)

IF t_out<0 THEN data1floor[2].7:=1; ELSE data1floor[2].7:=0; END_IF
data1floor[3]:=ABS(REAL_TO_BYTE(t_out));
data2floor[8]:=ABS(REAL_TO_BYTE(t_out));

winter;
t_max:=70;
t_min:=20;
IF t_out<15 THEN

	IF t_tambur > t_max THEN (*вимкнути колектор, якщо підлога тепліша за верхню межу температури*)
		freshbar_col:=FALSE;
	ELSE
		IF t_tambur< t_min THEN (*увімкнути колектор, якщо підлога холодніша за нижню межу*)
			freshbar_col:=TRUE;
		ELSE
			freshbar_col:= FALSE; (*ПОСТАВИТИ В ЗАЛЕЖНІСТЬ ВІД ЗОВНІШНЬОЇ ТЕМПЕРАТУРИ*)
		END_IF
	END_IF

	IF t_su > t_max THEN
		su_col_pidloga:=FALSE;
		su_col_stina:=FALSE;
			serverna_col:=FALSE;
	ELSE
		IF t_su< t_min THEN
			su_col_pidloga:=TRUE;
			su_col_stina:=TRUE;
			serverna_col:=TRUE;
		ELSE
			su_col_pidloga:=FALSE; (*ПОСТАВИТИ В ЗАЛЕЖНІСТЬ ВІД ЗОВНІШНЬОЇ ТЕМПЕРАТУРИ*)
			su_col_stina:=FALSE;
			serverna_col:=FALSE;
		END_IF
	END_IF

	IF t_spalnya>t_max THEN (*щоб не вистигала підлога*)
		spalnya_col:=FALSE;
	ELSE
		IF t_spalnya<t_min THEN
			spalnya_col:=TRUE;
		ELSE
			spalnya_col:=SPALNYA_HVAC.tepla_pidloga;
		END_IF
	END_IF


END_IF


IF VITALNYA_HVAC.heat_mode='OFF' THEN
				VITALNYA_HVAC.fancoil_speed:=0;
				(*VITALNYA_HVAC.collector:=2#00000000; all closed*)
				VITALNYA_HVAC.klapan:=16#7FFF;(*full closed*)
				VITALNYA_HVAC.zaslinka:=TRUE;(*closed*)
	END_IF

	IF KINO_HVAC.heat_mode='OFF'THEN
				KINO_HVAC.fancoil_speed:=0;
				(*KINO_HVAC.collector:=2#00000000; all closed*)
				KINO_HVAC.klapan:=16#7FFF;(*full closed*)
				KINO_HVAC.zaslinka:=TRUE;(*closed*)
	END_IF

	IF STUDIO_HVAC.heat_mode='OFF'THEN
				STUDIO_HVAC.fancoil_speed:=0;
				(*STUDIO_HVAC.collector:=2#00000000; all closed*)
				STUDIO_HVAC.klapan:=16#7FFF;(*full closed*)
				STUDIO_HVAC.zaslinka:=TRUE;(*closed*)
	END_IF

	IF KABINET_HVAC.heat_mode='OFF'THEN
				KABINET_HVAC.fancoil_speed:=0;
				(*KABINET_HVAC.collector:=2#00000000; all closed*)
				KABINET_HVAC.klapan:=16#7FFF;(*full closed*)
				KABINET_HVAC.zaslinka:=TRUE;(*closed*)
	END_IF

	IF DYTJACHA_HVAC.heat_mode='OFF'THEN
				DYTJACHA_HVAC.fancoil_speed:=0;
				(*DYTJACHA_HVAC.collector:=2#00000000; all closed*)
				DYTJACHA_HVAC.klapan:=16#7FFF;(*full closed*)
				DYTJACHA_HVAC.zaslinka:=TRUE;(*closed*)
	END_IF

	IF SPALNYA_HVAC.heat_mode='OFF'THEN
				SPALNYA_HVAC.fancoil_speed:=0;
				(*SPALNYA_HVAC.collector:=2#00000000; all closed*)
				SPALNYA_HVAC.klapan:=16#7FFF;(*full closed*)
				SPALNYA_HVAC.zaslinka:=TRUE;(*closed*)
	END_IF

(*__---_____
__---_____*)


data1floor[3]:=REAL_TO_BYTE (t_out);
data2floor[8]:=REAL_TO_BYTE (t_out);
(*локальні змінні для фенкойлів 3го поверхну об'явлені в області виходів*)

(*------------------------fancoil speed --------------------------------------------------*)
CASE DYTJACHA_HVAC.fancoil_speed OF
	0:	fancoil_dytjacha_low:=FALSE;
		fancoil_dytjacha_med:=FALSE;
		fancoil_dytjacha_high:=FALSE;

	1:	fancoil_dytjacha_low:=TRUE;
		fancoil_dytjacha_med:=FALSE;
		fancoil_dytjacha_high:=FALSE;

	2:	fancoil_dytjacha_low:=FALSE;
		fancoil_dytjacha_med:=TRUE;
		fancoil_dytjacha_high:=FALSE;

	3:	fancoil_dytjacha_low:=FALSE;
		fancoil_dytjacha_med:=FALSE;
		fancoil_dytjacha_high:=TRUE;
END_CASE

CASE SPALNYA_HVAC.fancoil_speed OF
	0:	fancoil_spalnya_low:=FALSE;
		fancoil_spalnya_med:=FALSE;
		fancoil_spalnya_high:=FALSE;

	1:	fancoil_spalnya_low:=TRUE;
		fancoil_spalnya_med:=FALSE;
		fancoil_spalnya_high:=FALSE;

	2:	fancoil_spalnya_low:=FALSE;
		fancoil_spalnya_med:=TRUE;
		fancoil_spalnya_high:=FALSE;

	3:	fancoil_spalnya_low:=FALSE;
		fancoil_spalnya_med:=FALSE;
		fancoil_spalnya_high:=TRUE;
END_CASE
CASE KABINET_HVAC.fancoil_speed OF
	0:	data2floor[0].0:=0; (*запис в масив даних, що відправляються на 2й поверх*)
		data2floor[0].1:=0;
		data2floor[0].2:=0;

	1:	data2floor[0].0:=1; (*запис в масив даних, що відправляються на 2й поверх*)
		data2floor[0].1:=0;
		data2floor[0].2:=0;

	2:	data2floor[0].0:=0; (*запис в масив даних, що відправляються на 2й поверх*)
		data2floor[0].1:=1;
		data2floor[0].2:=0;

	3:	data2floor[0].0:=0; (*запис в масив даних, що відправляються на 2й поверх*)
		data2floor[0].1:=0;
		data2floor[0].2:=1;
END_CASE

CASE KINO_HVAC.fancoil_speed OF
	0:	data2floor[0].3:=0; (*запис в масив даних, що відправляються на 2й поверх*)
		data2floor[0].4:=0;
		data2floor[0].5:=0;

	1:	data2floor[0].3:=1; (*запис в масив даних, що відправляються на 2й поверх*)
		data2floor[0].4:=0;
		data2floor[0].5:=0;

	2:	data2floor[0].3:=0; (*запис в масив даних, що відправляються на 2й поверх*)
		data2floor[0].4:=1;
		data2floor[0].5:=0;

	3:	data2floor[0].3:=0; (*запис в масив даних, що відправляються на 2й поверх*)
		data2floor[0].4:=0;
		data2floor[0].5:=1;
END_CASE

CASE VITALNYA_HVAC.fancoil_speed OF
	0:	data1floor[0].0:=0; (*запис в масив даних, що відправляються на 1й поверх*)
		data1floor[0].1:=0;
		data1floor[0].2:=0;

	1:	data1floor[0].0:=1; (*запис в масив даних, що відправляються на 1й поверх*)
		data1floor[0].1:=0;
		data1floor[0].2:=0;

	2:	data1floor[0].0:=0; (*запис в масив даних, що відправляються на 1й поверх*)
		data1floor[0].1:=1;
		data1floor[0].2:=0;

	3:	data1floor[0].0:=0; (*запис в масив даних, що відправляються на 1й поверх*)
		data1floor[0].1:=0;
		data1floor[0].2:=1;
END_CASE

(*--------------------------------------klapany--------------------------------------------*)
(*data1floor[2]:=WORD_TO_BYTE(VITALNYA_HVAC.klapan); data1floor[3]:=WORD_TO_BYTE(SHR(VITALNYA_HVAC.klapan,8));*)
klapan_vitalnya:=VITALNYA_HVAC.klapan;
klapan_spalnya:=SPALNYA_HVAC.klapan;
klapan_dytjacha:=DYTJACHA_HVAC.klapan;

data2floor[2]:=WORD_TO_BYTE(KABINET_HVAC.klapan); data2floor[3]:=WORD_TO_BYTE(SHR(KABINET_HVAC.klapan,8));
data2floor[4]:=WORD_TO_BYTE(KINO_HVAC.klapan); data2floor[5]:=WORD_TO_BYTE(SHR(KINO_HVAC.klapan,8));

(*------------------------------zaslinky------------------------------------*)
z_vitalnya:=VITALNYA_HVAC.zaslinka;
z_kabinet:=KABINET_HVAC.zaslinka;
z_kino:=KINO_HVAC.zaslinka;
z_dytjacha:=DYTJACHA_HVAC.zaslinka;
z_spalnya:=SPALNYA_HVAC.zaslinka;

(*-----------------------------tepla pidloga-------------------------------*)
data1floor[0].4:=VITALNYA_HVAC.tepla_pidloga;
data2floor[1].0:=KABINET_HVAC.tepla_pidloga;
data2floor[1].1:=KABINET_HVAC.tepla_pidloga;
data2floor[1].2:=STUDIO_HVAC.tepla_pidloga;
data2floor[1].3:=STUDIO_HVAC.tepla_pidloga;

dytjacha_col:=DYTJACHA_HVAC.tepla_pidloga;
spalnya_col:=SPALNYA_HVAC.tepla_pidloga;
END_PROGRAM
ACTION init:
IF i=500 THEN
	t_tamburPrev:=t_tambur_sum/i;
	t_suPrev:=t_su_sum/i;
	t_spalnyaPrev:=t_spalnya_sum/i;
	t_outPrev:=t_out_sum/i;
	t_tambur_sum:=0;
	t_su_sum:=0;
	t_spalnya_sum:=0;
	t_out_sum:=0;
	i:=501;
ELSE
	t_tambur_sum:=t_tambur_sum+temp_tambur*0.1;
	t_su_sum:=t_su_sum+temp_su*0.1;
	t_spalnya_sum:=t_spalnya_sum+temp_spalnya*0.1;
	t_out_sum:=t_out_sum+iT_out*0.1;
	i:=i+1;
END_IF
END_ACTION

(* POU HVAC/winter, ST *)
PROGRAM winter
VAR

END_VAR
(*--------------------------VITALNYA---------------------------------------------------------------*)

	IF VITALNYA_HVAC.heat_mode='HEAT' THEN
				VITALNYA_HVAC.zaslinka:=TRUE;(*closed*)
				VITALNYA_HVAC.tepla_pidloga:=TRUE; (*all opened*)
		CASE VITALNYA_HVAC.heat_speed OF

			1:	VITALNYA_HVAC.fancoil_speed:=1;
				VITALNYA_HVAC.klapan:=16#3FFF;
			2:	VITALNYA_HVAC.fancoil_speed:=2;
				VITALNYA_HVAC.klapan:=16#5FFF;
			3:	VITALNYA_HVAC.fancoil_speed:=3;
				VITALNYA_HVAC.klapan:=16#7FFF;
		END_CASE
	END_IF

	IF VITALNYA_HVAC.heat_mode='COOL' THEN
				VITALNYA_HVAC.klapan:=16#0;(*full closed*)
				VITALNYA_HVAC.zaslinka:=FALSE;
				VITALNYA_HVAC.tepla_pidloga:=FALSE; (*all closed*)

			CASE VITALNYA_HVAC.heat_speed OF
			1:	VITALNYA_HVAC.fancoil_speed:=1;
			2:	VITALNYA_HVAC.fancoil_speed:=2;
			3:	VITALNYA_HVAC.fancoil_speed:=3;
		END_CASE
	END_IF

	IF VITALNYA_HVAC.heat_mode='FAN' THEN
		VITALNYA_HVAC.tepla_pidloga:=FALSE;
		IF heat.t_out<0 THEN VITALNYA_HVAC.klapan:=16#3FFF;(*30%*) ELSE VITALNYA_HVAC.klapan:=16#0;END_IF
		CASE VITALNYA_HVAC.heat_speed OF
			1:	VITALNYA_HVAC.fancoil_speed:=0;
				VITALNYA_HVAC.zaslinka:=TRUE;(*closed*)
				VITALNYA_HVAC.klapan:=16#0;(*full closed*)
			2:	VITALNYA_HVAC.fancoil_speed:=2;
				VITALNYA_HVAC.zaslinka:=FALSE;(*opened*)
			3:	VITALNYA_HVAC.fancoil_speed:=3;
				VITALNYA_HVAC.zaslinka:=FALSE;(*opened*)
		END_CASE
	END_IF



(*--------------------------KABINET---------------------------------------------------------------*)
(*реверс двигуна клапана*)

	IF KABINET_HVAC.heat_mode='HEAT' THEN
				KABINET_HVAC.zaslinka:=TRUE;(*closed*)
				KABINET_HVAC.tepla_pidloga:=TRUE; (*all opened*)
		CASE KABINET_HVAC.heat_speed OF

			1:	KABINET_HVAC.fancoil_speed:=1;
				KABINET_HVAC.klapan:=16#5FFF;
			2:	KABINET_HVAC.fancoil_speed:=2;
				KABINET_HVAC.klapan:=16#3FFF;
			3:	KABINET_HVAC.fancoil_speed:=3;
				KABINET_HVAC.klapan:=16#1FFF;
		END_CASE
	END_IF

	IF KABINET_HVAC.heat_mode='COOL' THEN
				KABINET_HVAC.klapan:=16#7FFF;(*full closed*)
				KABINET_HVAC.zaslinka:=FALSE;
				KABINET_HVAC.tepla_pidloga:=FALSE; (*all closed*)

			CASE KABINET_HVAC.heat_speed OF
			1:	KABINET_HVAC.fancoil_speed:=1;
			2:	KABINET_HVAC.fancoil_speed:=2;
			3:	KABINET_HVAC.fancoil_speed:=3;
		END_CASE
	END_IF

	IF KABINET_HVAC.heat_mode='FAN' THEN
		KABINET_HVAC.tepla_pidloga:=FALSE;
		IF heat.t_out<0 THEN KABINET_HVAC.klapan:=16#5FFF;(*30%*) ELSE KABINET_HVAC.klapan:=16#7FFF;END_IF
		CASE KABINET_HVAC.heat_speed OF
			1:	KABINET_HVAC.fancoil_speed:=0;
				KABINET_HVAC.zaslinka:=TRUE;(*closed*)
				KABINET_HVAC.klapan:=16#7FFF;(*full closed*)
			2:	KABINET_HVAC.fancoil_speed:=2;
				KABINET_HVAC.zaslinka:=FALSE;(*opened*)
			3:	KABINET_HVAC.fancoil_speed:=3;
				KABINET_HVAC.zaslinka:=FALSE;(*opened*)
		END_CASE
	END_IF



(*--------------------------KINO---------------------------------------------------------------*)
(*реверс двигуна клапана*)
	IF KINO_HVAC.heat_mode='HEAT' THEN
				KINO_HVAC.zaslinka:=TRUE;(*closed*)
				KINO_HVAC.tepla_pidloga:=TRUE; (*all opened*)
		CASE KINO_HVAC.heat_speed OF

			1:	KINO_HVAC.fancoil_speed:=1;
				KINO_HVAC.klapan:=16#5FFF;
			2:	KINO_HVAC.fancoil_speed:=2;
				KINO_HVAC.klapan:=16#3FFF;
			3:	KINO_HVAC.fancoil_speed:=3;
				KINO_HVAC.klapan:=16#1FFF;
		END_CASE
	END_IF

	IF KINO_HVAC.heat_mode='COOL' THEN
				KINO_HVAC.klapan:=16#0;(*full closed*)
				KINO_HVAC.zaslinka:=FALSE;
				KINO_HVAC.tepla_pidloga:=FALSE; (*all closed*)

			CASE KINO_HVAC.heat_speed OF
			1:	KINO_HVAC.fancoil_speed:=1;
			2:	KINO_HVAC.fancoil_speed:=2;
			3:	KINO_HVAC.fancoil_speed:=3;
		END_CASE
	END_IF

	IF KINO_HVAC.heat_mode='FAN' THEN
		KINO_HVAC.tepla_pidloga:=FALSE;
		IF heat.t_out<0 THEN KINO_HVAC.klapan:=16#5FFF;(*30%*) ELSE KINO_HVAC.klapan:=16#7FFF;END_IF
		CASE KINO_HVAC.heat_speed OF
			1:	KINO_HVAC.fancoil_speed:=0;
				KINO_HVAC.zaslinka:=TRUE;(*closed*)
				KINO_HVAC.klapan:=16#7FFF;(*full closed*)
			2:	KINO_HVAC.fancoil_speed:=2;
				KINO_HVAC.zaslinka:=FALSE;(*opened*)
			3:	KINO_HVAC.fancoil_speed:=3;
				KINO_HVAC.zaslinka:=FALSE;(*opened*)
		END_CASE
	END_IF



(*--------------------------DYTJACHA---------------------------------------------------------------*)
(*реверс двигуна клапана*)
	IF DYTJACHA_HVAC.heat_mode='HEAT' THEN
				DYTJACHA_HVAC.zaslinka:=TRUE;(*closed*)
				DYTJACHA_HVAC.tepla_pidloga:=TRUE; (*all opened*)
		CASE DYTJACHA_HVAC.heat_speed OF

			1:	DYTJACHA_HVAC.fancoil_speed:=1;
				DYTJACHA_HVAC.klapan:=16#5FFF;
			2:	DYTJACHA_HVAC.fancoil_speed:=2;
				DYTJACHA_HVAC.klapan:=16#3FFF;
			3:	DYTJACHA_HVAC.fancoil_speed:=3;
				DYTJACHA_HVAC.klapan:=16#1FFF;
		END_CASE
	END_IF

	IF DYTJACHA_HVAC.heat_mode='COOL' THEN
				DYTJACHA_HVAC.klapan:=16#7FFF;(*full closed*)
				DYTJACHA_HVAC.zaslinka:=FALSE;
				DYTJACHA_HVAC.tepla_pidloga:=FALSE; (*all closed*)

			CASE DYTJACHA_HVAC.heat_speed OF
			1:	DYTJACHA_HVAC.fancoil_speed:=1;
			2:	DYTJACHA_HVAC.fancoil_speed:=2;
			3:	DYTJACHA_HVAC.fancoil_speed:=3;
		END_CASE
	END_IF

	IF DYTJACHA_HVAC.heat_mode='FAN' THEN
		DYTJACHA_HVAC.tepla_pidloga:=FALSE;
		IF heat.t_out<0 THEN DYTJACHA_HVAC.klapan:=16#5FFF;(*30%*) ELSE DYTJACHA_HVAC.klapan:=16#7FFF;END_IF
		CASE DYTJACHA_HVAC.heat_speed OF
			1:	DYTJACHA_HVAC.fancoil_speed:=0;
				DYTJACHA_HVAC.zaslinka:=TRUE;(*closed*)
				DYTJACHA_HVAC.klapan:=16#7FFF;(*full closed*)
			2:	DYTJACHA_HVAC.fancoil_speed:=2;
				DYTJACHA_HVAC.zaslinka:=FALSE;(*opened*)
			3:	DYTJACHA_HVAC.fancoil_speed:=3;
				DYTJACHA_HVAC.zaslinka:=FALSE;(*opened*)
		END_CASE
	END_IF



(*--------------------------SPALNYA---------------------------------------------------------------*)

	IF SPALNYA_HVAC.heat_mode='HEAT' THEN
				SPALNYA_HVAC.zaslinka:=TRUE;(*closed*)
				SPALNYA_HVAC.tepla_pidloga:=TRUE; (*all opened*)
		CASE SPALNYA_HVAC.heat_speed OF

			1:	SPALNYA_HVAC.fancoil_speed:=1;
				SPALNYA_HVAC.klapan:=16#3FFF;
			2:	SPALNYA_HVAC.fancoil_speed:=2;
				SPALNYA_HVAC.klapan:=16#5FFF;
			3:	SPALNYA_HVAC.fancoil_speed:=3;
				SPALNYA_HVAC.klapan:=16#7FFF;
		END_CASE
	END_IF

	IF SPALNYA_HVAC.heat_mode='COOL' THEN
				SPALNYA_HVAC.klapan:=16#0;(*full closed*)
				SPALNYA_HVAC.zaslinka:=FALSE;
				SPALNYA_HVAC.tepla_pidloga:=FALSE; (*all closed*)

			CASE SPALNYA_HVAC.heat_speed OF
			1:	SPALNYA_HVAC.fancoil_speed:=1;
			2:	SPALNYA_HVAC.fancoil_speed:=2;
			3:	SPALNYA_HVAC.fancoil_speed:=3;
		END_CASE
	END_IF

	IF SPALNYA_HVAC.heat_mode='FAN' THEN
		SPALNYA_HVAC.tepla_pidloga:=FALSE;
		IF heat.t_out<0 THEN SPALNYA_HVAC.klapan:=16#3FFF;(*30%*) ELSE SPALNYA_HVAC.klapan:=16#0;END_IF
		CASE SPALNYA_HVAC.heat_speed OF
			1:	SPALNYA_HVAC.fancoil_speed:=0;
				SPALNYA_HVAC.zaslinka:=TRUE;(*closed*)
				SPALNYA_HVAC.klapan:=16#0;(*full closed*)
			2:	SPALNYA_HVAC.fancoil_speed:=2;
				SPALNYA_HVAC.zaslinka:=FALSE;(*opened*)
			3:	SPALNYA_HVAC.fancoil_speed:=3;
				SPALNYA_HVAC.zaslinka:=FALSE;(*opened*)
		END_CASE
	END_IF
END_PROGRAM

(* POU ADS_write, ST *)
PROGRAM ADS_write
VAR
	write_timeout: TIME;
	b_write1, b_write2: BOOL;
	write_ads1, write_ads2: ADSWRITE;

	timer1, timer2:TP;
	errorcounter1, errorcounter2, pack_c:CTU ;
	test_word: WORD;
	i,j,i1,j1: INT;
	data_changed: BOOL;
	try_again2, try_again1: BOOL;
	temp: INT;
END_VAR
write_timeout:=t#3s;


FOR i:=0 TO (SIZEOF(data2floor))-1 DO
	IF data2floor[i]<>data2floor_prev[i] THEN
		b_write2:=TRUE;
		EXIT;
	ELSE
		b_write2:=FALSE;
	END_IF
END_FOR




IF write_ads2.BUSY THEN b_write2:=FALSE; END_IF

	write_ads2(
		NETID:=ads_adr2,
		PORT:=800,
		IDXGRP:=16#4020,
		IDXOFFS:=0,
		WRITE:=b_write2,
		TMOUT:=write_timeout,
		LEN:=SIZEOF(data2floor),
		SRCADDR:=ADR(data2floor));

IF write_ads2.ERR AND NOT timer2.Q THEN
	timer2.IN:=TRUE;
	try_again2:=TRUE;
END_IF
timer2(PT:=write_timeout);
timer2.IN:=FALSE;

FOR j:=0 TO (SIZEOF(data2floor))-1 DO
	data2floor_prev[j]:=data2floor[j];
END_FOR

(*1floor*)
FOR i1:=0 TO (SIZEOF(data1floor))-1 DO
	IF data1floor[i1]<>data1floor_prev[i1] THEN
		b_write1:=TRUE;
		EXIT;
	ELSE
		b_write1:=FALSE;
	END_IF
END_FOR

IF try_again1 AND NOT timer1.Q THEN
	b_write1:=TRUE;
	try_again1:=FALSE;
END_IF


IF write_ads1.BUSY THEN b_write1:=FALSE; END_IF

	write_ads1(
		NETID:=ads_adr1,
		PORT:=800,
		IDXGRP:=16#4020,
		IDXOFFS:=0,
		WRITE:=b_write1,
		TMOUT:=write_timeout,
		LEN:=SIZEOF(data1floor),
		SRCADDR:=ADR(data1floor));

IF write_ads1.ERR AND NOT timer1.Q THEN
	timer1.IN:=TRUE;
	try_again1:=TRUE;
END_IF
timer1(PT:=write_timeout);
timer1.IN:=FALSE;


FOR j1:=0 TO (SIZEOF(data1floor))-1 DO
	data1floor_prev[j1]:=data1floor[j1];
END_FOR
END_PROGRAM

(* POU HVAC/summer, ST *)
PROGRAM summer
VAR

END_VAR
data1floor[0].3:=TRUE

(*--------------------------VITALNYA---------------------------------------------------------------*)

	IF VITALNYA_HVAC.heat_mode='HEAT' THEN
				VITALNYA_HVAC.zaslinka:=TRUE;(*closed*)
				VITALNYA_HVAC.tepla_pidloga:=TRUE; (*all opened*)
		CASE VITALNYA_HVAC.heat_speed OF

			1:	VITALNYA_HVAC.fancoil_speed:=1;
				VITALNYA_HVAC.klapan:=16#3FFF;
			2:	VITALNYA_HVAC.fancoil_speed:=2;
				VITALNYA_HVAC.klapan:=16#5FFF;
			3:	VITALNYA_HVAC.fancoil_speed:=3;
				VITALNYA_HVAC.klapan:=16#7FFF;
		END_CASE
	END_IF

	IF VITALNYA_HVAC.heat_mode='COOL' THEN
				VITALNYA_HVAC.klapan:=16#0;(*full closed*)
				VITALNYA_HVAC.zaslinka:=FALSE;
				VITALNYA_HVAC.tepla_pidloga:=FALSE; (*all closed*)

			CASE VITALNYA_HVAC.heat_speed OF
			1:	VITALNYA_HVAC.fancoil_speed:=1;
			2:	VITALNYA_HVAC.fancoil_speed:=2;
			3:	VITALNYA_HVAC.fancoil_speed:=3;
		END_CASE
	END_IF

	IF VITALNYA_HVAC.heat_mode='FAN' THEN
		VITALNYA_HVAC.tepla_pidloga:=FALSE;
		IF heat.t_out<0 THEN VITALNYA_HVAC.klapan:=16#3FFF;(*30%*) ELSE VITALNYA_HVAC.klapan:=16#0;END_IF
		CASE VITALNYA_HVAC.heat_speed OF
			1:	VITALNYA_HVAC.fancoil_speed:=0;
				VITALNYA_HVAC.zaslinka:=TRUE;(*closed*)
				VITALNYA_HVAC.klapan:=16#0;(*full closed*)
			2:	VITALNYA_HVAC.fancoil_speed:=2;
				VITALNYA_HVAC.zaslinka:=FALSE;(*opened*)
			3:	VITALNYA_HVAC.fancoil_speed:=3;
				VITALNYA_HVAC.zaslinka:=FALSE;(*opened*)
		END_CASE
	END_IF



(*--------------------------KABINET---------------------------------------------------------------*)
(*реверс двигуна клапана*)

	IF KABINET_HVAC.heat_mode='HEAT' THEN
				KABINET_HVAC.zaslinka:=TRUE;(*closed*)
				KABINET_HVAC.tepla_pidloga:=TRUE; (*all opened*)
		CASE KABINET_HVAC.heat_speed OF

			1:	KABINET_HVAC.fancoil_speed:=1;
				KABINET_HVAC.klapan:=16#5FFF;
			2:	KABINET_HVAC.fancoil_speed:=2;
				KABINET_HVAC.klapan:=16#3FFF;
			3:	KABINET_HVAC.fancoil_speed:=3;
				KABINET_HVAC.klapan:=16#1FFF;
		END_CASE
	END_IF

	IF KABINET_HVAC.heat_mode='COOL' THEN
				KABINET_HVAC.klapan:=16#7FFF;(*full closed*)
				KABINET_HVAC.zaslinka:=FALSE;
				KABINET_HVAC.tepla_pidloga:=FALSE; (*all closed*)

			CASE KABINET_HVAC.heat_speed OF
			1:	KABINET_HVAC.fancoil_speed:=1;
			2:	KABINET_HVAC.fancoil_speed:=2;
			3:	KABINET_HVAC.fancoil_speed:=3;
		END_CASE
	END_IF

	IF KABINET_HVAC.heat_mode='FAN' THEN
		KABINET_HVAC.tepla_pidloga:=FALSE;
		IF heat.t_out<0 THEN KABINET_HVAC.klapan:=16#5FFF;(*30%*) ELSE KABINET_HVAC.klapan:=16#7FFF;END_IF
		CASE KABINET_HVAC.heat_speed OF
			1:	KABINET_HVAC.fancoil_speed:=0;
				KABINET_HVAC.zaslinka:=TRUE;(*closed*)
				KABINET_HVAC.klapan:=16#7FFF;(*full closed*)
			2:	KABINET_HVAC.fancoil_speed:=2;
				KABINET_HVAC.zaslinka:=FALSE;(*opened*)
			3:	KABINET_HVAC.fancoil_speed:=3;
				KABINET_HVAC.zaslinka:=FALSE;(*opened*)
		END_CASE
	END_IF



(*--------------------------KINO---------------------------------------------------------------*)
(*реверс двигуна клапана*)
	IF KINO_HVAC.heat_mode='HEAT' THEN
				KINO_HVAC.zaslinka:=TRUE;(*closed*)
				KINO_HVAC.tepla_pidloga:=TRUE; (*all opened*)
		CASE KINO_HVAC.heat_speed OF

			1:	KINO_HVAC.fancoil_speed:=1;
				KINO_HVAC.klapan:=16#5FFF;
			2:	KINO_HVAC.fancoil_speed:=2;
				KINO_HVAC.klapan:=16#3FFF;
			3:	KINO_HVAC.fancoil_speed:=3;
				KINO_HVAC.klapan:=16#1FFF;
		END_CASE
	END_IF

	IF KINO_HVAC.heat_mode='COOL' THEN
				KINO_HVAC.klapan:=16#0;(*full closed*)
				KINO_HVAC.zaslinka:=FALSE;
				KINO_HVAC.tepla_pidloga:=FALSE; (*all closed*)

			CASE KINO_HVAC.heat_speed OF
			1:	KINO_HVAC.fancoil_speed:=1;
			2:	KINO_HVAC.fancoil_speed:=2;
			3:	KINO_HVAC.fancoil_speed:=3;
		END_CASE
	END_IF

	IF KINO_HVAC.heat_mode='FAN' THEN
		KINO_HVAC.tepla_pidloga:=FALSE;
		IF heat.t_out<0 THEN KINO_HVAC.klapan:=16#5FFF;(*30%*) ELSE KINO_HVAC.klapan:=16#7FFF;END_IF
		CASE KINO_HVAC.heat_speed OF
			1:	KINO_HVAC.fancoil_speed:=0;
				KINO_HVAC.zaslinka:=TRUE;(*closed*)
				KINO_HVAC.klapan:=16#7FFF;(*full closed*)
			2:	KINO_HVAC.fancoil_speed:=2;
				KINO_HVAC.zaslinka:=FALSE;(*opened*)
			3:	KINO_HVAC.fancoil_speed:=3;
				KINO_HVAC.zaslinka:=FALSE;(*opened*)
		END_CASE
	END_IF



(*--------------------------DYTJACHA---------------------------------------------------------------*)
(*реверс двигуна клапана*)
	IF DYTJACHA_HVAC.heat_mode='HEAT' THEN
				DYTJACHA_HVAC.zaslinka:=TRUE;(*closed*)
				DYTJACHA_HVAC.tepla_pidloga:=TRUE; (*all opened*)
		CASE DYTJACHA_HVAC.heat_speed OF

			1:	DYTJACHA_HVAC.fancoil_speed:=1;
				DYTJACHA_HVAC.klapan:=16#5FFF;
			2:	DYTJACHA_HVAC.fancoil_speed:=2;
				DYTJACHA_HVAC.klapan:=16#3FFF;
			3:	DYTJACHA_HVAC.fancoil_speed:=3;
				DYTJACHA_HVAC.klapan:=16#1FFF;
		END_CASE
	END_IF

	IF DYTJACHA_HVAC.heat_mode='COOL' THEN
				DYTJACHA_HVAC.klapan:=16#7FFF;(*full closed*)
				DYTJACHA_HVAC.zaslinka:=FALSE;
				DYTJACHA_HVAC.tepla_pidloga:=FALSE; (*all closed*)

			CASE DYTJACHA_HVAC.heat_speed OF
			1:	DYTJACHA_HVAC.fancoil_speed:=1;
			2:	DYTJACHA_HVAC.fancoil_speed:=2;
			3:	DYTJACHA_HVAC.fancoil_speed:=3;
		END_CASE
	END_IF

	IF DYTJACHA_HVAC.heat_mode='FAN' THEN
		DYTJACHA_HVAC.tepla_pidloga:=FALSE;
		IF heat.t_out<0 THEN DYTJACHA_HVAC.klapan:=16#5FFF;(*30%*) ELSE DYTJACHA_HVAC.klapan:=16#7FFF;END_IF
		CASE DYTJACHA_HVAC.heat_speed OF
			1:	DYTJACHA_HVAC.fancoil_speed:=0;
				DYTJACHA_HVAC.zaslinka:=TRUE;(*closed*)
				DYTJACHA_HVAC.klapan:=16#7FFF;(*full closed*)
			2:	DYTJACHA_HVAC.fancoil_speed:=2;
				DYTJACHA_HVAC.zaslinka:=FALSE;(*opened*)
			3:	DYTJACHA_HVAC.fancoil_speed:=3;
				DYTJACHA_HVAC.zaslinka:=FALSE;(*opened*)
		END_CASE
	END_IF



(*--------------------------SPALNYA---------------------------------------------------------------*)

	IF SPALNYA_HVAC.heat_mode='HEAT' THEN
				SPALNYA_HVAC.zaslinka:=TRUE;(*closed*)
				SPALNYA_HVAC.tepla_pidloga:=TRUE; (*all opened*)
		CASE SPALNYA_HVAC.heat_speed OF

			1:	SPALNYA_HVAC.fancoil_speed:=1;
				SPALNYA_HVAC.klapan:=16#3FFF;
			2:	SPALNYA_HVAC.fancoil_speed:=2;
				SPALNYA_HVAC.klapan:=16#5FFF;
			3:	SPALNYA_HVAC.fancoil_speed:=3;
				SPALNYA_HVAC.klapan:=16#7FFF;
		END_CASE
	END_IF

	IF SPALNYA_HVAC.heat_mode='COOL' THEN
				SPALNYA_HVAC.klapan:=16#0;(*full closed*)
				SPALNYA_HVAC.zaslinka:=FALSE;
				SPALNYA_HVAC.tepla_pidloga:=FALSE; (*all closed*)

			CASE SPALNYA_HVAC.heat_speed OF
			1:	SPALNYA_HVAC.fancoil_speed:=1;
			2:	SPALNYA_HVAC.fancoil_speed:=2;
			3:	SPALNYA_HVAC.fancoil_speed:=3;
		END_CASE
	END_IF

	IF SPALNYA_HVAC.heat_mode='FAN' THEN
		SPALNYA_HVAC.tepla_pidloga:=FALSE;
		IF heat.t_out<0 THEN SPALNYA_HVAC.klapan:=16#3FFF;(*30%*) ELSE SPALNYA_HVAC.klapan:=16#0;END_IF
		CASE SPALNYA_HVAC.heat_speed OF
			1:	SPALNYA_HVAC.fancoil_speed:=0;
				SPALNYA_HVAC.zaslinka:=TRUE;(*closed*)
				SPALNYA_HVAC.klapan:=16#0;(*full closed*)
			2:	SPALNYA_HVAC.fancoil_speed:=2;
				SPALNYA_HVAC.zaslinka:=FALSE;(*opened*)
			3:	SPALNYA_HVAC.fancoil_speed:=3;
				SPALNYA_HVAC.zaslinka:=FALSE;(*opened*)
		END_CASE
	END_IF
END_PROGRAM
